PROGRAM MAIN
VAR
	stop : BOOL;
	manualStep : BOOL := TRUE;
	manualSuction : BOOL;
	
	moduleWB : WoodBunkEx;
	moduleCIP : ChipboardEx;
	
	exec1 : BOOL;
	exec2 : BOOL;
END_VAR

CallHardware(); //start program with hardware call - pass values and arrays into function blocks
SetupHardware(); //initialize values

runModules(); //LLD

CallHardware(); //end program with hardware call

ACTION runModules:
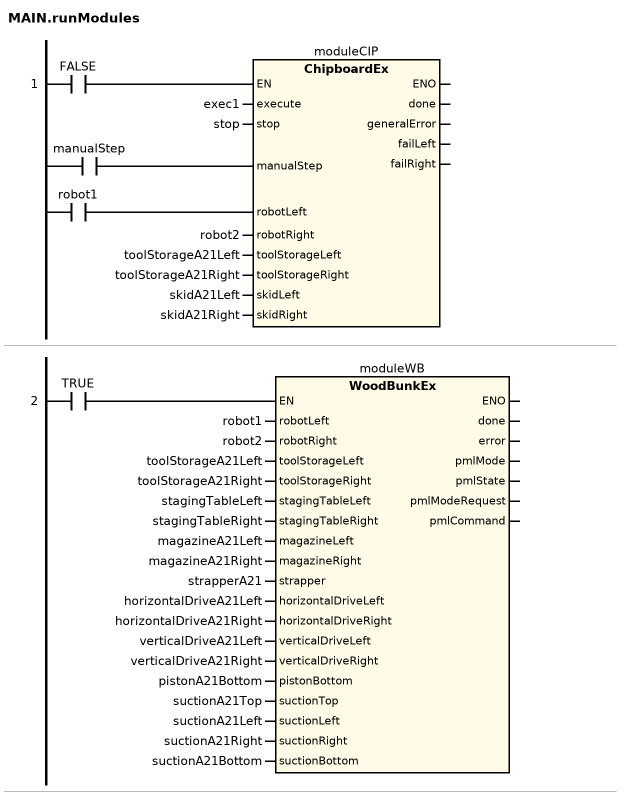
// NETWORK 1
IF FALSE THEN
    moduleCIP(
        execute := exec1,
        stop := stop,
        manualStep := manualStep,
        robotLeft := robot1,
        robotRight := robot2,
        toolStorageLeft := toolStorageA21Left,
        toolStorageRight := toolStorageA21Right,
        skidLeft := skidA21Left,
        skidRight := skidA21Right); // ChipboardEx
END_IF

// NETWORK 2
moduleWB(
    robotLeft := robot1,
    robotRight := robot2,
    toolStorageLeft := toolStorageA21Left,
    toolStorageRight := toolStorageA21Right,
    stagingTableLeft := stagingTableLeft,
    stagingTableRight := stagingTableRight,
    magazineLeft := magazineA21Left,
    magazineRight := magazineA21Right,
    strapper := strapperA21,
    horizontalDriveLeft := horizontalDriveA21Left,
    horizontalDriveRight := horizontalDriveA21Right,
    verticalDriveLeft := verticalDriveA21Left,
    verticalDriveRight := verticalDriveA21Right,
    pistonBottom := pistonA21Bottom,
    suctionTop := suctionA21Top,
    suctionLeft := suctionA21Left,
    suctionRight := suctionA21Right,
    suctionBottom := suctionA21Bottom); // WoodBunkEx
END_ACTION

END_PROGRAM

(* stored: Version 1.1.0.1, ProductVersion 3.1.4024.12
   POU MAIN: Id {9caf58b7-eccf-4a65-a3e3-2c8d81beb312}, SpecialFunc None
   Action runModules: Id {797c012e-5535-4cfd-a7fe-f38cfe08cb9f} *)
